// Mitsubishi GX Works2 project: d1 카운트   PLC: Q02/Q02H

PROGRAM MAIN
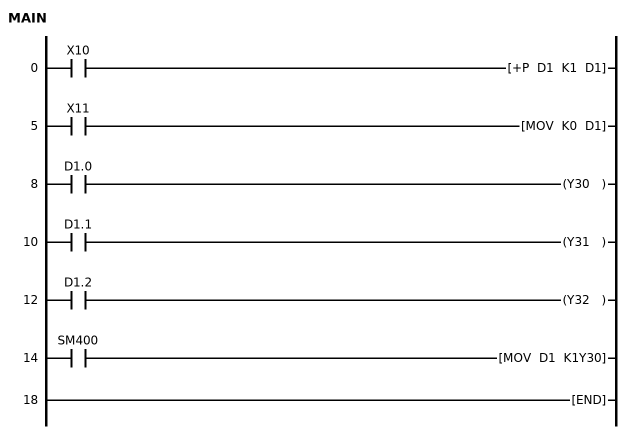
0     LD      X10
      +P      D1 K1 D1
5     LD      X11
      MOV     K0 D1
8     LD      D1.0
      OUT     Y30
10    LD      D1.1
      OUT     Y31
12    LD      D1.2
      OUT     Y32
14    LD      SM400
      MOV     D1 K1Y30
18    END
END_PROGRAM
